// TIA Portal V19 export
TYPE "TMeasuring_ERRORWORD"
// stored: Access Published
   STRUCT
      SystemFault : Bool;   // A
      ConfigFault : Bool;   // One of the the four SLS limits is active; operates together with bit 1
      UserFault : Bool;   // Error accessing a logical address
      CommandNotAccepted : Bool;   // Collect warnings
      PeripheralError : Bool;   // Equivalent Acc / Dec without jerk component
   END_STRUCT;
END_TYPE
